Staubli VAL3: onEditItem.pgx

public program onEditItem(string& x_sEvent[], num x_nIndex, num x_nIndexItem)
  local joint l_jJoint
  local num i
  local string l_sEmpty
  local string l_sMessage
begin
  // edit the custom element that was add in the list
  l_jJoint=jEditPoint.tData[x_nIndexItem].jJoint
  call use:findPos(x_sEvent,">",i)
  i=i+1
  // clean the line
  call use:listcursor(use:nView,false)
  l_sEmpty=""
  switch x_nIndex
    case 0
      //  j1-value
      if cycleStatus:bCycle
        // set a limit +- 5
        call use:changeValue(l_jJoint.j1,l_jJoint.j1-5,l_jJoint.j1+5,i+40-use:nBottomX,use:nView+1,l_sEmpty)
      else
        call use:changeValue(l_jJoint.j1,0,0,i+40-use:nBottomX,use:nView+1,l_sEmpty)
      endIf
    break
    case 1
      //  j2-value
      if cycleStatus:bCycle
        // set a limit +- 5
        call use:changeValue(l_jJoint.j2,l_jJoint.j2-5,l_jJoint.j2+5,i+40-use:nBottomX,use:nView+1,l_sEmpty)
      else
        call use:changeValue(l_jJoint.j2,0,0,i+40-use:nBottomX,use:nView+1,l_sEmpty)
      endIf
    break
    case 2
      //  j3-value
      if cycleStatus:bCycle
        // set a limit +- 5
        call use:changeValue(l_jJoint.j3,l_jJoint.j3-5,l_jJoint.j3+5,i+40-use:nBottomX,use:nView+1,l_sEmpty)
      else
        call use:changeValue(l_jJoint.j3,0,0,i+40-use:nBottomX,use:nView+1,l_sEmpty)
      endIf
    break
    case 3
      //  j4-value
      if cycleStatus:bCycle
        // set a limit +- 5
        call use:changeValue(l_jJoint.j4,l_jJoint.j4-5,l_jJoint.j4+5,i+40-use:nBottomX,use:nView+1,l_sEmpty)
      else
        call use:changeValue(l_jJoint.j4,0,0,i+40-use:nBottomX,use:nView+1,l_sEmpty)
      endIf
    break
    case 4
      //  j5-value
      if cycleStatus:bCycle
        // set a limit +- 5
        call use:changeValue(l_jJoint.j5,l_jJoint.j5-5,l_jJoint.j5+5,i+40-use:nBottomX,use:nView+1,l_sEmpty)
      else
        call use:changeValue(l_jJoint.j5,0,0,i+40-use:nBottomX,use:nView+1,l_sEmpty)
      endIf
    break
    case 5
      //  j6-value
      if cycleStatus:bCycle
        // set a limit +- 5
        call use:changeValue(l_jJoint.j6,l_jJoint.j6-5,l_jJoint.j6+5,i+40-use:nBottomX,use:nView+1,l_sEmpty)
      else
        call use:changeValue(l_jJoint.j6,0,0,i+40-use:nBottomX,use:nView+1,l_sEmpty)
      endIf
    break
  endSwitch
  //
  if isInRange(l_jJoint)
    jEditPoint.tData[x_nIndexItem].jJoint=l_jJoint
  else
    // error using the trsf
    call language:message(l_sMessage,-5)
    popUpMsg(l_sMessage)
  endIf
  // wait no key
  call use:nullKey(nKey)
end
